TYPE Array4Byte :
UNION
	arrByte			:ARRAY[0..3] OF BYTE;
	rValue			:INT;
END_UNION
END_TYPE

(* stored: Version 1.1.0.1
   DUT Array4Byte: Id {23a7f7d2-5e01-472c-b54e-623da5011b29} *)
